FUNCTION_BLOCK FB_TwinCat
VAR_INPUT
	input	:	BOOL;
	inputreal:	REAL;
END_VAR
VAR_OUTPUT
	outputreal			:	real;
END_VAR
VAR
END_VAR

IF input=TRUE THEN
	outputreal:=inputreal;
END_IF
//oder
IF 			input=FALSE THEN
	outputreal:=inputreal/2;
END_IF;

END_FUNCTION_BLOCK

(* stored: Version 1.1.0.1, ProductVersion 3.1.4024.9
   POU FB_TwinCat: Id {ddc5bf00-72ef-445b-b5e5-e6d1b5d2fc4b}, SpecialFunc None *)
